// TIA Portal V17 export
// export: Created 2024-09-02T12:50:34.9414674Z, ExportSetting WithDefaults, DisplayName Totally Integrated Automation Portal, DisplayVersion V17, DisplayName TIA Portal Openness, DisplayVersion V17, DisplayName TIA Portal Version Control Interface, DisplayVersion V17, DisplayName STEP 7 Professional, DisplayVersion V17, DisplayName STEP 7 Safety, DisplayVersion V17, DisplayName WinCC Professional, DisplayVersion V17
TYPE "typ_Key"
// stored: IsFailsafeCompliant false
   STRUCT
      KST_1 : Char;   // Kostenstelle / Cost centre
      KST_2 : Char;   // Kostenstelle / Cost centre
      KST_3 : Char;   // Kostenstelle / Cost centre
      KST_4 : Char;   // Kostenstelle / Cost centre
      EMP_NR_1 : Char;   // Mitarbeiter / Employees
      EMP_NR_2 : Char;   // Mitarbeiter / Employees
      EMP_NR_3 : Char;   // Mitarbeiter / Employees
      EMP_NR_4 : Char;   // Mitarbeiter / Employees
      PERMISSION : Char;   // Berechtigung / Permission
      YEAR : Byte;   // Zeitstempel / Time stamp
      MONTH : Byte;   // Zeitstempel / Time stamp
      DAY : Byte;   // Zeitstempel / Time stamp
      HOUR : Byte;   // Zeitstempel / Time stamp
      MINUTE : Byte;   // Zeitstempel / Time stamp
      SECOND : Byte;   // Zeitstempel / Time stamp
      FIRST_KST_1 : Char;   // Kostenstelle - Erstwert / Cost center - initial value
      FIRST_KST_2 : Char;   // Kostenstelle - Erstwert / Cost center - initial value
      FIRST_KST_3 : Char;   // Kostenstelle - Erstwert / Cost center - initial value
      FIRST_KST_4 : Char;   // Kostenstelle - Erstwert / Cost center - initial value
      FIRST_EMP_NR_1 : Char;   // Mitarbeiter - Erstwert / Employees - first value
      FIRST_EMP_NR_2 : Char;   // Mitarbeiter - Erstwert / Employees - first value
      FIRST_EMP_NR_3 : Char;   // Mitarbeiter - Erstwert / Employees - first value
      FIRST_EMP_NR_4 : Char;   // Mitarbeiter - Erstwert / Employees - first value
      FIRST_PERMISSION : Char;   // Berechtigung - Erstwert / Permission - First value
      FIRST_YEAR : Byte;   // Zeitstempel - Erstwert / Timestamp - First value
      FIRST_MONTH : Byte;   // Zeitstempel - Erstwert / Timestamp - First value
      FIRST_DAY : Byte;   // Zeitstempel - Erstwert / Timestamp - First value
      FIRST_HOUR : Byte;   // Zeitstempel - Erstwert / Timestamp - First value
      FIRST_MINUTE : Byte;   // Zeitstempel - Erstwert / Timestamp - First value
      FIRST_SECOND : Byte;   // Zeitstempel - Erstwert / Timestamp - First value
   END_STRUCT;
END_TYPE
